TYPE U_MOVE_DATA :
UNION
  stData              : ARRAY[1..MAX_MOVER] OF ST_MOVE_DATA;

  byData    AT %I*    : ARRAY[1..MAX_MOVER] OF
                        ARRAY[1..SIZEOF(ST_MOVE_DATA)] OF BYTE;
END_UNION
END_TYPE

(* stored: Version 1.1.0.1, ProductVersion 3.1.4026.12
   DUT U_MOVE_DATA: Id {7b10e0c0-017b-4551-9e37-6791ab3e1721} *)
